{attribute 'GeneratedUsingTerminal: ELX3312-0000-0016'}
{attribute addProperty BoxType "ELX3312-0000-0016"}
{attribute addProperty Id "TC_Inputs_Channel_1AT %I*TC_Inputs_Channel_4A3944819TC_Inputs_Channel_2AT %I*TC_Inputs_Channel_4A3944819WcStateAT %I*WcState_9091E0EB2InfoDataAT %I*InfoData_94A18F5E2"}
{attribute addProperty CRC "3866174781"}
{attribute addProperty Size "22"}
TYPE ELX3312_E671253D EXTENDS EtcSlaveTerminalBase_947E5A46 :
STRUCT
	{attribute addProperty Name "TC_Inputs_Channel_1"}
	TC_Inputs_Channel_1 : TC_Inputs_Channel_4A394481;
	{attribute addProperty Name "TC_Inputs_Channel_2"}
	TC_Inputs_Channel_2 : TC_Inputs_Channel_4A394481;
	{attribute addProperty Name "WcState"}
	WcState : WcState_9091E0EB;
	{attribute addProperty Name "InfoData"}
	InfoData : InfoData_94A18F5E;
END_STRUCT
END_TYPE

(* stored: Version 1.2.0.0, ProductVersion 3.1.4024.9
   DUT ELX3312_E671253D: Id {06909a76-3134-4cfe-b027-26e001405120} *)
